FUNCTION_BLOCK FB_Example
VAR
    x : INT := zz;
END_VAR
BEGIN
END_FUNCTION_BLOCK
